# EPICS substitutions: apps/xpsMotorApp/Db/hpsTargetScan.substitutions
file "$(TOP)/db/XPSAuxAi.db"
{
pattern
{         P,         R,       PORT,CHAN,   LOPR,  HOPR,  PREC,     SCAN  }
{US1-2-BOT:, XPSAuxAi0,  US1-2-BOT, 0,    -10.0,  10.0,  3,    "1 second"}
{US1-2-BOT:, XPSAuxAi1,  US1-2-BOT, 1,    -10.0,  10.0,  3,    "1 second"}
{US1-2-BOT:, XPSAuxAi2,  US1-2-BOT, 2,    -10.0,  10.0,  3,    "1 second"}
{US1-2-BOT:, XPSAuxAi3,  US1-2-BOT, 3,    -10.0,  10.0,  3,    "1 second"}
}
